FUNCTION_BLOCK FB_PU_Schuetz
VAR_IN_OUT
END_VAR
VAR_INPUT
	Freigabe_auto			: BOOL;
	Freigabe_Deakt_auto		: BOOL;
	Betrieb_Anford_auto		: BOOL;
	Quittierung				: BOOL;
	Parameter_init			: ST_PU_Schuetz_Parameter;
END_VAR
VAR_OUTPUT
	{attribute 'OPC.UA.DA' := '1'}Steuerung				: ST_PU_Schuetz_Steuerung;			
	{attribute 'OPC.UA.DA' := '1'}Stellwert				: ST_PU_Schuetz_Stellwert;			
	{attribute 'OPC.UA.DA' := '1'}Zustand					: ST_PU_Schuetz_Zustand;		
	{attribute 'OPC.UA.DA' := '1'}Parameter				: ST_PU_Schuetz_Parameter;			
END_VAR
VAR
	Zustandscheck			: FB_PU_Schuetz_Zustandscheck;
	Logik					: FB_PU_Schuetz_Logik;
	Ablaufsteuerung			: FB_PU_Schuetz_Ablaufsteuerung;
	QuitTrig					: FB_SetResetFallTrigger;

	SchreibeDaten			: FB_PU_Schuetz_Output;
	OUT_Stellung			AT %Q* : BOOL;
END_VAR

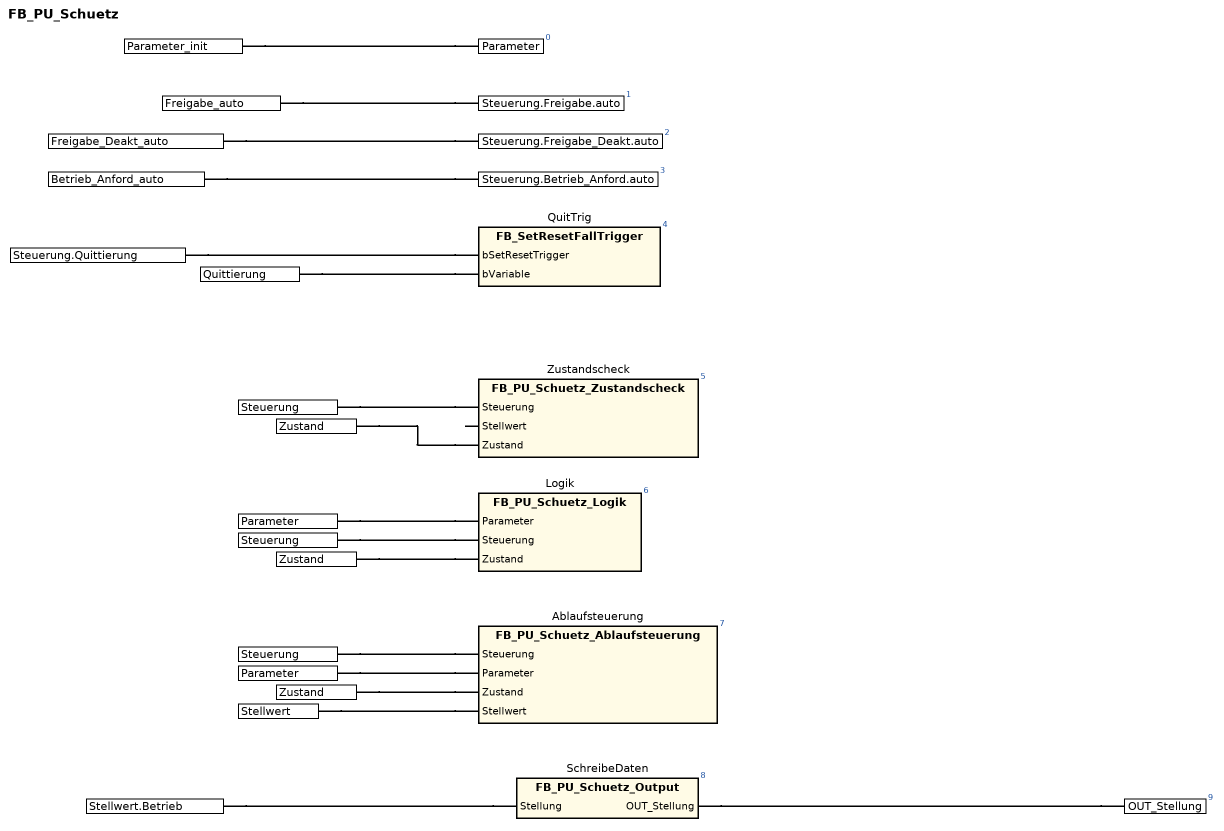
Parameter := Parameter_init;
Steuerung.Freigabe.auto := Freigabe_auto;
Steuerung.Freigabe_Deakt.auto := Freigabe_Deakt_auto;
Steuerung.Betrieb_Anford.auto := Betrieb_Anford_auto;
QuitTrig(bSetResetTrigger := Steuerung.Quittierung, bVariable := Quittierung); // FB_SetResetFallTrigger
Zustandscheck(Steuerung := Steuerung, Zustand := Zustand); // FB_PU_Schuetz_Zustandscheck
Logik(Parameter := Parameter, Steuerung := Steuerung, Zustand := Zustand); // FB_PU_Schuetz_Logik
Ablaufsteuerung(Steuerung := Steuerung, Parameter := Parameter, Zustand := Zustand, Stellwert := Stellwert); // FB_PU_Schuetz_Ablaufsteuerung
SchreibeDaten(Stellung := Stellwert.Betrieb); // FB_PU_Schuetz_Output
OUT_Stellung := SchreibeDaten.OUT_Stellung;

END_FUNCTION_BLOCK

(* stored: Version 1.1.0.1, ProductVersion 3.1.4024.9
   POU FB_PU_Schuetz: Id {03c6f6e3-4f96-4f9d-8f3e-307e29ea41ee}, SpecialFunc None *)
